(* IEC 61131-3 sources: horner-cscape-mcp/artifacts/projects/Fail_SyntaxNearSemi_Location_Proj/pous, 1 file *)

(* ---- POU_SyntaxNearSemi.st ---- *)
PROGRAM POU_SyntaxNearSemi
VAR
    TankLevel : REAL := 50.0;
    TargetLevel : REAL := 60.0;
END_VAR

TargetLevel := TankLevel + ;
END_PROGRAM
